GLOBALCONSTANTS DefaultPool_PWM12_Bargraph (* Bargraph geometry and scale constants (Length, ScalePx, Min, Max, Type) *)
  PACKAGE Uebungen::const::UT::PWM12;
  VAR_GLOBAL CONSTANT
    Bargraph_PWM_Q01_ScalePx : REAL := 0.0072834799;
    Bargraph_PWM_Q01_LengthPx : REAL := 468.0;
    Bargraph_PWM_Q01_Min : REAL := 0.0;
    Bargraph_PWM_Q01_Max : REAL := 64255.0;
    Bargraph_PWM_Q01_Type : USINT := 3;
    Bargraph_PWM_Q02_ScalePx : REAL := 0.0072834799;
    Bargraph_PWM_Q02_LengthPx : REAL := 468.0;
    Bargraph_PWM_Q02_Min : REAL := 0.0;
    Bargraph_PWM_Q02_Max : REAL := 64255.0;
    Bargraph_PWM_Q02_Type : USINT := 3;
    Bargraph_PWM_Q03_ScalePx : REAL := 0.0072834799;
    Bargraph_PWM_Q03_LengthPx : REAL := 468.0;
    Bargraph_PWM_Q03_Min : REAL := 0.0;
    Bargraph_PWM_Q03_Max : REAL := 64255.0;
    Bargraph_PWM_Q03_Type : USINT := 3;
    Bargraph_PWM_Q04_ScalePx : REAL := 0.0072834799;
    Bargraph_PWM_Q04_LengthPx : REAL := 468.0;
    Bargraph_PWM_Q04_Min : REAL := 0.0;
    Bargraph_PWM_Q04_Max : REAL := 64255.0;
    Bargraph_PWM_Q04_Type : USINT := 3;
    Bargraph_PWM_Q05_ScalePx : REAL := 0.0072834799;
    Bargraph_PWM_Q05_LengthPx : REAL := 468.0;
    Bargraph_PWM_Q05_Min : REAL := 0.0;
    Bargraph_PWM_Q05_Max : REAL := 64255.0;
    Bargraph_PWM_Q05_Type : USINT := 3;
    Bargraph_PWM_Q06_ScalePx : REAL := 0.0072834799;
    Bargraph_PWM_Q06_LengthPx : REAL := 468.0;
    Bargraph_PWM_Q06_Min : REAL := 0.0;
    Bargraph_PWM_Q06_Max : REAL := 64255.0;
    Bargraph_PWM_Q06_Type : USINT := 3;
    Bargraph_PWM_Q07_ScalePx : REAL := 0.0072834799;
    Bargraph_PWM_Q07_LengthPx : REAL := 468.0;
    Bargraph_PWM_Q07_Min : REAL := 0.0;
    Bargraph_PWM_Q07_Max : REAL := 64255.0;
    Bargraph_PWM_Q07_Type : USINT := 3;
    Bargraph_PWM_Q08_ScalePx : REAL := 0.0072834799;
    Bargraph_PWM_Q08_LengthPx : REAL := 468.0;
    Bargraph_PWM_Q08_Min : REAL := 0.0;
    Bargraph_PWM_Q08_Max : REAL := 64255.0;
    Bargraph_PWM_Q08_Type : USINT := 3;
    Bargraph_PWM_Q09_ScalePx : REAL := 0.0072834799;
    Bargraph_PWM_Q09_LengthPx : REAL := 468.0;
    Bargraph_PWM_Q09_Min : REAL := 0.0;
    Bargraph_PWM_Q09_Max : REAL := 64255.0;
    Bargraph_PWM_Q09_Type : USINT := 3;
    Bargraph_PWM_Q10_ScalePx : REAL := 0.0072834799;
    Bargraph_PWM_Q10_LengthPx : REAL := 468.0;
    Bargraph_PWM_Q10_Min : REAL := 0.0;
    Bargraph_PWM_Q10_Max : REAL := 64255.0;
    Bargraph_PWM_Q10_Type : USINT := 3;
    Bargraph_PWM_Q11_ScalePx : REAL := 0.0072834799;
    Bargraph_PWM_Q11_LengthPx : REAL := 468.0;
    Bargraph_PWM_Q11_Min : REAL := 0.0;
    Bargraph_PWM_Q11_Max : REAL := 64255.0;
    Bargraph_PWM_Q11_Type : USINT := 3;
    Bargraph_PWM_Q12_ScalePx : REAL := 0.0072834799;
    Bargraph_PWM_Q12_LengthPx : REAL := 468.0;
    Bargraph_PWM_Q12_Min : REAL := 0.0;
    Bargraph_PWM_Q12_Max : REAL := 64255.0;
    Bargraph_PWM_Q12_Type : USINT := 3;
  END_VAR
END_GLOBALCONSTANTS
